PROGRAM MAIN
VAR
    bLampa  AT %Q* : BOOL; // To jest nasza dioda
    fbTimer : TON;         // Timer do mrugania
END_VAR

fbTimer(IN := NOT fbTimer.Q, PT := T#999MS); // Czekaj 0.5 sekundy

IF fbTimer.Q THEN
    bLampa := NOT bLampa; // Zmień stan diody na przeciwny
END_IF

END_PROGRAM

(* stored: Version 1.1.0.1, ProductVersion 3.1.4024.16
   POU MAIN: Id {9d920f35-5d14-420b-82cb-73a41417625b}, SpecialFunc None *)
